(* IEC 61131-3 sources: mocks/src, 4 files *)

(* ---- OffDelayMock_false.st ---- *)
NAMESPACE Siemens.Ax.Mocks
    FUNCTION_BLOCK OffDelayMock_false
        VAR
            iecTimer : ARRAY[0..27] of BYTE;
        END_VAR
        VAR_INPUT
            duration : LTIME;
            signal : BOOL;
        END_VAR
        VAR_OUTPUT
            output : BOOL;
            elapsedTime : LTIME;
        END_VAR
        output := FALSE;
    END_FUNCTION_BLOCK
END_NAMESPACE

(* ---- OffDelayMock_true.st ---- *)
NAMESPACE Siemens.Ax.Mocks
    FUNCTION_BLOCK OffDelayMock_true
        VAR
            iecTimer : ARRAY[0..27] of BYTE;
        END_VAR
        VAR_INPUT
            duration : LTIME;
            signal : BOOL;
        END_VAR
        VAR_OUTPUT
            output : BOOL;
            elapsedTime : LTIME;
        END_VAR
        output := TRUE;
    END_FUNCTION_BLOCK
END_NAMESPACE

(* ---- OnDelayMock_false.st ---- *)
NAMESPACE Siemens.Ax.Mocks
    FUNCTION_BLOCK OnDelayMock_false
        VAR
            iecTimer : ARRAY[0..27] of BYTE;
        END_VAR
        VAR_INPUT
            duration : LTIME;
            signal : BOOL;
        END_VAR
        VAR_OUTPUT
            output : BOOL;
            elapsedTime : LTIME;
        END_VAR
        output := FALSE;
    END_FUNCTION_BLOCK
END_NAMESPACE

(* ---- OnDelayMock_true.st ---- *)
NAMESPACE Siemens.Ax.Mocks
    FUNCTION_BLOCK OnDelayMock_true
        VAR
            iecTimer : ARRAY[0..27] of BYTE;
        END_VAR
        VAR_INPUT
            duration : LTIME;
            signal : BOOL;
        END_VAR
        VAR_OUTPUT
            output : BOOL;
            elapsedTime : LTIME;
        END_VAR
        output := TRUE;
    END_FUNCTION_BLOCK
END_NAMESPACE
